FUNCTION_BLOCK FB_RegulMoteur
VAR_INPUT
		Consigne: LREAL;					//sets the desired speed of the Motor in rot/min
		lrValeurDirection: LREAL;			//the converted value from Tachymeter with Direction added
		xDirection: BOOL;					//Forward or Backward
		xOnOff: BOOL;						//Motor On or Off
		PARA : ST_CTRL_PID_PARAMS;			//Parameters for the PID
		xReset: BOOL;						//Reset the PID-Block
		PID : FB_CTRL_PID;					//PID-Block
		fbConvertNumToMotorOut : FB_Qa;		//Convert the PID-Output into numeric values send to the motor
		fbConvertTachoToNumSpeed : FB_Ia;	//Convert the numeric values from the Tachymeter into rot/min
		TimerOffAlarm : UINT;				//after enabling the Motor all Alarms will be blocked for 2sec
END_VAR
VAR_OUTPUT
	xError : BOOL;							//Error state
	iErrorID : INT;							//Error ID
END_VAR

//convert Tacho speed into rot/min
fbConvertTachoToNumSpeed();

//call the PID-Block if needed
IF xOnOff THEN
	PID(fOut=>fbConvertNumToMotorOut.lrConsigne,fSetpointValue:=Consigne,
		fActualValue:=fbConvertTachoToNumSpeed.lrValeur,eMode:=2,stParams:=PARA);
	//decrese the delay for alarms
	IF TimerOffAlarm>0 THEN
		TimerOffAlarm:=TimerOffAlarm-1;
	END_IF
ELSE
	fbConvertNumToMotorOut.lrConsigne:=0;
	TimerOffAlarm:=200; //200 @ 10ms Cycle --> 2sec
END_IF

//Convert now to have the value as fast as possible written to the motor
fbConvertNumToMotorOut();

//Reset the PID block
IF xReset THEN
	PID.bSync:=xReset;
END_IF


//******************************************
//Output actions
//******************************************

//Error management
IF PID.bError AND xOnOff AND TimerOffAlarm=0 THEN
xError:=TRUE;
iErrorID:=300;
ELSIF PID.bARWactive AND xOnOff AND TimerOffAlarm=0 THEN
	xError:=TRUE;
	iErrorId:=301;
ELSE
	xError:=FALSE;
END_IF

END_FUNCTION_BLOCK

(* stored: Version 1.1.0.1, ProductVersion 3.1.4020.6
   POU FB_RegulMoteur: Id {76bd808d-6760-4a61-a5ed-d48ddecd1ecc}, SpecialFunc None *)
